FUNCTION_BLOCK Sensor
VAR
END_VAR

PROPERTY PUBLIC Triggered : BOOL
GET
END_GET
END_PROPERTY

END_FUNCTION_BLOCK

(* stored: Version 1.1.0.1
   POU Sensor: Id {536536a2-3df6-4334-8e4c-d88ca9b76854}, SpecialFunc None
   Property Triggered: Id {d2992bb6-0f90-4c42-9df9-3b231c5afb70}
   Get Get: Id {09fec3f4-a157-4aab-84de-4dc875f2921a} *)
